FUNCTION_BLOCK Disturbance (* Basic Function Block Type *)
  (* Standard: 61499-2 *)
  (* Version 0.0, 2011-12-23, 4DIAC-IDE, 4DIAC-Consortium *)
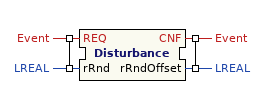
  EVENT_INPUT
    REQ WITH rRnd; (* Normal Execution Request *)
  END_EVENT
  EVENT_OUTPUT
    CNF WITH rRndOffset; (* Execution Confirmation *)
  END_EVENT
  VAR_INPUT
    rRnd : LREAL; (* Input event qualifier *)
  END_VAR
  VAR_OUTPUT
    rRndOffset : LREAL := 0; (* Output event qualifier *)
  END_VAR
  VAR
    rRndScale : LREAL := 0.1; (* Internal Variable *)
  END_VAR
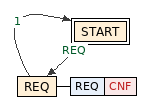
  EC_STATES
    START; (* Initial State *)
    REQ : REQ -> CNF; (* Normal execution *)
  END_STATES
  EC_TRANSITIONS
    START TO REQ := REQ;
    REQ TO START := 1;
  END_TRANSITIONS
  ALGORITHM REQ IN ST: (* Normally executed algorithm *)
rRndOffset:=rRndOffset + (rRnd-0.5)*rRndScale;
IF rRndOffset>=1 THEN
	rRndOffset:=1;
ELSE
	IF rRndOffset<=-1 THEN
		rRndOffset:=-1;
	END_IF;
END_IF;
  END_ALGORITHM
END_FUNCTION_BLOCK
